Fanuc KAREL source: NC0011.KL

-- PROVISIONAL review KL for V940-1; original PC SHA256 144e36a330c7a4e505eacad9600bb4a7957f30d60f172c259a383748ace0f8b5
-- Incomplete behavior may be omitted. Consult companion uncertainty JSON. Do not deploy.
PROGRAM NC0011
%NOLOCKGROUP
-- UNRESOLVED_LOCAL_POOL 1 cells at code offset 3; source declarations unknown
-- DIRECT_LOCAL_WORD_ACCESS alone does not prove INTEGER, REAL, or BOOLEAN
BEGIN
  -- V9_EXPOSED_INDEXED_TABLE_HINT layout=0001; 40 counted words exposed once; source arms/runtime held
  -- V9_CONDITION_STACK_HINT 20 bounded expression windows; static native code-base-relative target link; source arms held
  -- UNRESOLVED_PC offsets 0-8; opcodes 2B,2C,7B
  -- UNRESOLVED_PC offsets 13-20; opcodes 9D,23
  -- UNRESOLVED_PC offsets 25-38; opcodes 21,9D,57,79
  -- UNRESOLVED_PC offsets 43-56; opcodes 21,9D,57,79
  -- UNRESOLVED_PC offsets 61-74; opcodes 21,9D,57,79
  -- UNRESOLVED_PC offsets 79-92; opcodes 21,9D,57,79
  -- UNRESOLVED_PC offsets 97-110; opcodes 21,9D,57,79
  -- UNRESOLVED_PC offsets 115-128; opcodes 21,9D,57,79
  -- UNRESOLVED_PC offsets 133-146; opcodes 21,9D,57,79
  -- UNRESOLVED_PC offsets 151-164; opcodes 21,9D,57,79
  -- UNRESOLVED_PC offsets 169-182; opcodes 21,9D,57,79
  -- UNRESOLVED_PC offsets 187-200; opcodes 21,9D,57,79
  -- UNRESOLVED_PC offsets 205-218; opcodes 21,9D,57,79
  -- UNRESOLVED_PC offsets 223-236; opcodes 21,9D,57,79
  -- UNRESOLVED_PC offsets 241-254; opcodes 21,9D,57,79
  -- UNRESOLVED_PC offsets 259-272; opcodes 21,9D,57,79
  -- UNRESOLVED_PC offsets 277-290; opcodes 21,9D,57,79
  -- UNRESOLVED_PC offsets 295-308; opcodes 21,9D,57,79
  -- UNRESOLVED_PC offsets 313-326; opcodes 21,9D,57,79
  -- UNRESOLVED_PC offsets 331-344; opcodes 21,9D,57,79
  -- UNRESOLVED_PC offsets 349-362; opcodes 21,9D,57,79
  -- UNRESOLVED_PC offsets 367-380; opcodes 21,9D,57,79
  -- UNRESOLVED_PC offsets 385-399; opcodes 21,9D,52,23
  -- UNRESOLVED_PC offsets 404-409; opcodes 7A
  -- UNRESOLVED_PC offsets 414-432; opcodes 21,2E,52,23
  -- UNRESOLVED_PC offsets 442-447; opcodes 7A
  -- UNRESOLVED_PC offsets 452-470; opcodes 21,2E,52,23
  -- UNRESOLVED_PC offsets 480-485; opcodes 7A
  -- UNRESOLVED_PC offsets 490-508; opcodes 21,2E,52,23
  -- UNRESOLVED_PC offsets 518-523; opcodes 7A
  -- UNRESOLVED_PC offsets 528-546; opcodes 21,2E,52,23
  -- UNRESOLVED_PC offsets 556-561; opcodes 7A
  -- UNRESOLVED_PC offsets 566-584; opcodes 21,2E,52,23
  -- UNRESOLVED_PC offsets 594-599; opcodes 7A
  -- UNRESOLVED_PC offsets 604-622; opcodes 21,2E,52,23
  -- UNRESOLVED_PC offsets 632-637; opcodes 7A
  -- UNRESOLVED_PC offsets 642-660; opcodes 21,2E,52,23
  -- UNRESOLVED_PC offsets 670-675; opcodes 7A
  -- UNRESOLVED_PC offsets 680-698; opcodes 21,2E,52,23
  -- UNRESOLVED_PC offsets 708-713; opcodes 7A
  -- UNRESOLVED_PC offsets 718-736; opcodes 21,2E,52,23
  -- UNRESOLVED_PC offsets 746-751; opcodes 7A
  -- UNRESOLVED_PC offsets 756-774; opcodes 21,2E,52,23
  -- UNRESOLVED_PC offsets 784-789; opcodes 7A
  -- UNRESOLVED_PC offsets 794-812; opcodes 21,2E,52,23
  -- UNRESOLVED_PC offsets 822-827; opcodes 7A
  -- UNRESOLVED_PC offsets 832-850; opcodes 21,2E,52,23
  -- UNRESOLVED_PC offsets 860-865; opcodes 7A
  -- UNRESOLVED_PC offsets 870-888; opcodes 21,2E,52,23
  -- UNRESOLVED_PC offsets 898-903; opcodes 7A
  -- UNRESOLVED_PC offsets 908-926; opcodes 21,2E,52,23
  -- UNRESOLVED_PC offsets 936-941; opcodes 7A
  -- UNRESOLVED_PC offsets 946-964; opcodes 21,2E,52,23
  -- UNRESOLVED_PC offsets 974-979; opcodes 7A
  -- UNRESOLVED_PC offsets 984-1002; opcodes 21,2E,52,23
  -- UNRESOLVED_PC offsets 1012-1017; opcodes 7A
  -- UNRESOLVED_PC offsets 1022-1040; opcodes 21,2E,52,23
  -- UNRESOLVED_PC offsets 1050-1055; opcodes 7A
  -- UNRESOLVED_PC offsets 1060-1078; opcodes 21,2E,52,23
  -- UNRESOLVED_PC offsets 1088-1093; opcodes 7A
  -- UNRESOLVED_PC offsets 1098-1116; opcodes 21,2E,52,23
  -- UNRESOLVED_PC offsets 1126-1131; opcodes 7A
  -- UNRESOLVED_PC offsets 1136-1154; opcodes 21,2E,52,23
  -- UNRESOLVED_PC offsets 1164-1168; opcodes 7F
  -- UNRESOLVED_PC offsets 1173-1177; opcodes 27,AA
  -- UNRESOLVED_PC offsets 1182-1186; opcodes 7F
END NC0011
